Yaskawa INFORM job: compressor_cylinder_program.JBI

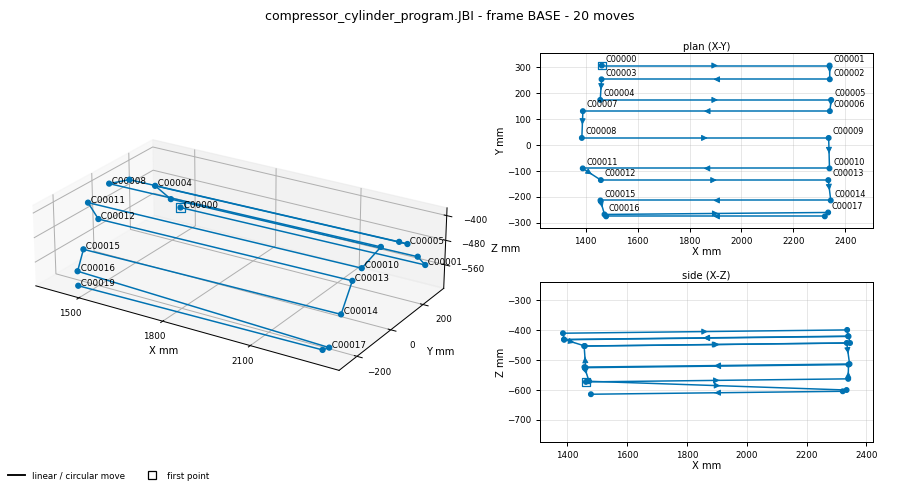
[picture p0: tool path of compressor_cylinder_program.JBI in frame BASE, 20 of 23 moves have a stored position in this frame; points joined in program order, loops and branches not executed]
/JOB
//NAME compressor_cylinder_program
//POS
///NPOS 20,0,20,0,0,0
///TOOL 0
///POSTYPE BASE
///RECTAN
///RCONF 0,0,0,0,0,0,0,0,0,0,0,0,0,0,0,0,0,0,0,0,0,0,0,0
C00000=1461.900613,306.418041,-572.812061,-175.000000,-60.000000,-89.788582
C00001=2339.554084,306.418067,-562.576872,-175.000000,-60.000000,-89.788582
C00002=2340.429535,253.314952,-514.873579,175.000000,-52.801105,-89.492834
C00003=1461.002935,253.314926,-525.129446,175.000000,-52.801105,-89.492834
C00004=1455.917090,173.895381,-452.975741,-175.000000,-31.762251,-88.920679
C00005=2345.637556,173.895407,-442.599827,-175.000000,-31.762251,-88.920679
C00006=2340.683816,130.652074,-420.604159,157.714803,-5.000000,5.000000
C00007=1389.033078,130.652046,-431.702304,157.714803,-5.000000,5.000000
C00008=1385.048919,27.440052,-409.914062,175.000000,-5.000000,5.000000
C00009=2336.021444,27.440080,-398.823827,175.000000,-5.000000,5.000000
C00010=2339.196650,-89.918508,-419.680547,-158.203651,-5.000000,-5.000000
C00011=1388.488053,-89.918536,-430.767704,-158.203651,-5.000000,-5.000000
C00012=1458.337724,-135.022906,-452.661333,175.000000,-31.656128,88.916201
C00013=2334.653111,-135.022880,-442.441749,175.000000,-31.656128,88.916201
C00014=2344.055286,-213.422125,-512.893508,175.000000,-52.325433,89.484038
C00015=1456.796513,-213.422152,-523.240714,175.000000,-52.325433,89.484038
C00016=1472.386641,-267.365754,-570.707293,175.000000,-60.000000,89.777894
C00017=2334.151319,-259.707891,-599.945123,-175.000000,-71.612958,89.777894
C00018=2321.219990,-274.701408,-604.213213,175.000000,-60.000000,89.990693
C00019=1478.603809,-274.701433,-614.039797,175.000000,-60.000000,89.990693
///POSTYPE PULSE
///PULSE
EX00000=89088.0
///POSTYPE PULSE
///PULSE
EC00000=89088.0
EC00001=89088.0
EC00002=89088.0
EC00003=89088.0
EC00004=89088.0
EC00005=89088.0
EC00006=89088.0
EC00007=89088.0
EC00008=89088.0
EC00009=89088.0
EC00010=89088.0
EC00011=89088.0
EC00012=89088.0
EC00013=89088.0
EC00014=89088.0
EC00015=89088.0
EC00016=89088.0
EC00017=89088.0
EC00018=89088.0
EC00019=89088.0
//INST
///DATE 2023/08/16 14:18
///ATTR SC,RW,RJ
////FRAME BASE
///GROUP1 RB1,ST1
NOP
MOVJ P009 EX000 VJ=15.00
MOVJ C00000 EC00000 VJ=15.0
CALL JOB:SPYON
MOVL C00001 EC00001 V=150.0
MOVL C00002 EC00002 V=150.0
MOVL C00003 EC00003 V=150.0
MOVL C00004 EC00004 V=150.0
MOVL C00005 EC00005 V=150.0
MOVL C00006 EC00006 V=150.0
MOVL C00007 EC00007 V=150.0
MOVL C00008 EC00008 V=150.0
MOVL C00009 EC00009 V=150.0
MOVL C00010 EC00010 V=150.0
MOVL C00011 EC00011 V=150.0
MOVL C00012 EC00012 V=150.0
MOVL C00013 EC00013 V=150.0
MOVL C00014 EC00014 V=150.0
MOVL C00015 EC00015 V=150.0
MOVL C00016 EC00016 V=150.0
MOVL C00017 EC00017 V=150.0
MOVL C00018 EC00018 V=150.0
MOVL C00019 EC00019 V=150.0
CALL JOB:SPYOF
MOVJ P009 VJ=15.00
MOVL P009 EX00000 V=150.0
END
